{attribute 'linkalways'} 
{attribute 'no_explicit_call' := 'This FB is a CLASS and must be accessed using methods or properties'}
{attribute 'enable_dynamic_creation'}
FUNCTION_BLOCK Node_F_VN_AddToContainerElements_TcVnPoint3_LREAL EXTENDS VisionNode
VAR
    aValue : _TcVnPoint3_LREAL;
    ipContainer : _ITcVnContainer;
    hrPrev : _HRESULT(S_OK);
    hresult : _HRESULT(S_OK);
END_VAR

METHOD PUBLIC  Clone : I_Node
VAR
    pNode : POINTER TO Node_F_VN_AddToContainerElements_TcVnPoint3_LREAL;
END_VAR
pNode := __NEW(Node_F_VN_AddToContainerElements_TcVnPoint3_LREAL);
Clone := pNode^;
END_METHOD

METHOD FB_init : BOOL
VAR_INPUT
    bInitRetains : BOOL; // if TRUE, the retain variables are initialized (warm start / cold start)
    bInCopyCode : BOOL;  // if TRUE, the instance afterwards gets moved into the copy code (online change)
END_VAR
AddInput('aValue', aValue);
AddInput('ipContainer', ipContainer);
AddInput('hrPrev', hrPrev);
AddOutput('ipContainer', ipContainer);
AddOutput('hresult',hresult);
END_METHOD

METHOD PROTECTED OnExecute : HRESULT
hresult.Value := F_VN_AddToContainerElements_TcVnPoint3_LREAL(
    aValue := aValue.Value,
    ipContainer := ipContainer.Value,
    hrPrev:= hrPrev.Value);
END_METHOD

METHOD PUBLIC PreExecutionCheck
VAR_INPUT
    Check : I_PreExecutionChecks;
END_VAR
Check.IsTrue(ipContainer.IsValid, 'ipContainer must be a valid container');
Check.IsTrue(ipContainer.HasType(TC_GLOBAL_CONST_LIST.ContainerType_Vector_TcVnPoint3_LREAL), 'ipContainer contains incorrect type');
END_METHOD

END_FUNCTION_BLOCK

(* stored: Version 1.1.0.1, ProductVersion 3.1.4024.13
   POU Node_F_VN_AddToContainerElements_TcVnPoint3_LREAL: Id {dea7d249-e3ad-4ce5-a668-1061b840fd63}, SpecialFunc None
   Folder Constructor: Id {89749a01-2b23-4df4-8167-4d4a45b0e69b}
   Method Clone: Id {8ee950b3-2873-4739-9d52-b2c87e1b4136}
   Method FB_init: Id {46a0e59c-ed5e-4f7e-8add-6014151aa54b}
   Method OnExecute: Id {ad7276d4-1a75-4415-b89f-478be293dd66}
   Method PreExecutionCheck: Id {b6789a4f-1e4a-4695-9127-bf012554aa94} *)
